FUNCTION_BLOCK ABSTRACT HardwareNode EXTENDS Node

METHOD PUBLIC Clone : I_Node
VAR
END_VAR
Clone := THIS^;
END_METHOD

METHOD Dispose
VAR_INPUT
END_VAR
END_METHOD

END_FUNCTION_BLOCK

(* stored: Version 1.1.0.1, ProductVersion 3.1.4024.13
   POU HardwareNode: Id {8a18619e-3bff-0ee0-18d6-780ce4fc0c54}, SpecialFunc None
   Method Clone: Id {cec82d75-f155-4784-a43d-387f9ee1bdac}
   Method Dispose: Id {7708a250-3ac6-4df8-aaf2-fad4b0369d75} *)
